FUNCTION_BLOCK Calc_Spiral_Linear_Move
  (* Standard: 61499-2 *)
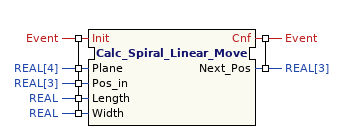
  EVENT_INPUT
    Init WITH Plane, Pos_in, Length, Width;
  END_EVENT
  EVENT_OUTPUT
    Cnf WITH Next_Pos;
  END_EVENT
  VAR_INPUT
    Plane : ARRAY [0..3] OF REAL;
    Pos_in : ARRAY [0..2] OF REAL;
    Length : REAL := 0;
    Width : REAL := 0;
  END_VAR
  VAR_OUTPUT
    Next_Pos : ARRAY [0..2] OF REAL;
  END_VAR
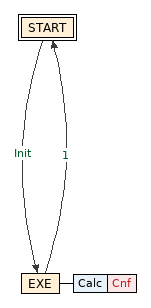
  EC_STATES
    START;
    EXE : Calc -> Cnf;
  END_STATES
  EC_TRANSITIONS
    EXE TO START := 1;
    START TO EXE := Init;
  END_TRANSITIONS
  ALGORITHM Calc IN Lua:

			local zoff = (Plane[4] - Plane[2]*(Pos_in[2] + Width) - Plane[1]*(Pos_in[1] + Length))/Plane[3]
			Next_Pos = {Pos_in[1] + Length, Pos_in[2] + Width, zoff}
  END_ALGORITHM
END_FUNCTION_BLOCK
